{attribute addProperty BoxType "CU1124-0000-0016"}
{attribute addProperty Id "A_0004_CU1128_0000_0000A_0004_CU1128_0000_0000_277E4A76992124"}
{attribute addProperty CRC "1337575023"}
{attribute addProperty SizeInBites "992"}
{attribute addProperty SizeInBytes "124"}
TYPE A_0003_CU1124_0000_0016_4FB9C66F EXTENDS CU1124_179A0949 :
STRUCT
	{attribute addProperty Name "A_0004_CU1128_0000_0000"}
	A_0004_CU1128_0000_0000 : A_0004_CU1128_0000_0000_277E4A76;
END_STRUCT
END_TYPE

(* stored: Version 1.2.0.0, ProductVersion 3.1.4024.9
   DUT A_0003_CU1124_0000_0016_4FB9C66F: Id {99bf408b-6431-4948-bdba-66d7abe700af} *)
